# EPICS alarm handler configuration: mps_database/bareTest/alarms/areas/mpln_unds_mp07.alhConfig
GROUP NULL MPLN:UNDS:MP07:1
$ALIAS MPS Link Node 215
$GUIDANCE
LTUH MPS
   Group Name: MPLN:UNDS:MP07:1
   Summary PV:  MPLN:UNDS:MP07:1:STATSUMY
$END
CHANNEL  MPLN:UNDS:MP07:1    MPLN:UNDS:MP07:1:MPS_EN_RBV		-----
CHANNEL  MPLN:UNDS:MP07:1    MPLN:UNDS:MP07:1:LC1_MODE_RBV		-----
